TYPE ST_OperatorStationStatus :
STRUCT
    eState                  : E_OperatorExchangeState;
    eInstruction            : E_OperatorInstruction;
    bExchangeComplete       : BOOL;
    bIndexPermissive        : BOOL;
    bPartRemovedConfirmed   : BOOL;
    bRejectConfirmed        : BOOL;
    bRejectArmed            : BOOL;
    bRejectEdgeAccepted     : BOOL;
    bRejectWaitingForClear  : BOOL;
    bRejectPopupRequest     : BOOL;
    bPartPresent            : BOOL;
    bRejectChutePartPresent : BOOL;
    bResultValid            : BOOL;
    bResultPassed           : BOOL;
    sMessage                : STRING(255);
    bPbupPresent : BOOL;
    bLoadSetComplete : BOOL;
    bMissingPbup : BOOL;
    bMissingProduct : BOOL;
    bMissingPbupAlert : BOOL;
    bMissingProductAlert : BOOL;
END_STRUCT
END_TYPE

(* stored: Version 1.1.0.1, ProductVersion 3.1.4026.18
   DUT ST_OperatorStationStatus: Id {648bab67-1c7c-45e5-8d7e-abeb87bda2b3} *)
